{attribute 'strict'}
TYPE E_FixtureStateMeasurement :
(
	FIXTURE_MEASUREMENT_START 				:= 0,
	FIXTURE_MEASUREMENT_WAIT_FOR_BUSY 		:= 10,
	FIXTURE_MEASUREMENT_WAIT_FOR_RESPONSE 	:= 20,
	FIXTURE_MEASUREMENT_REMEASUREMENT		:= 30,
	FIXTURE_MEASUREMENT_DONE				:= 40
);
END_TYPE

(* stored: Version 1.1.0.1, ProductVersion 3.1.4024.9
   DUT E_FixtureStateMeasurement: Id {bacdff6f-c2c7-40cd-b827-847d64bf7346} *)
